Universal Robots PolyScope program: 33-trigger_reduced_mode.urp

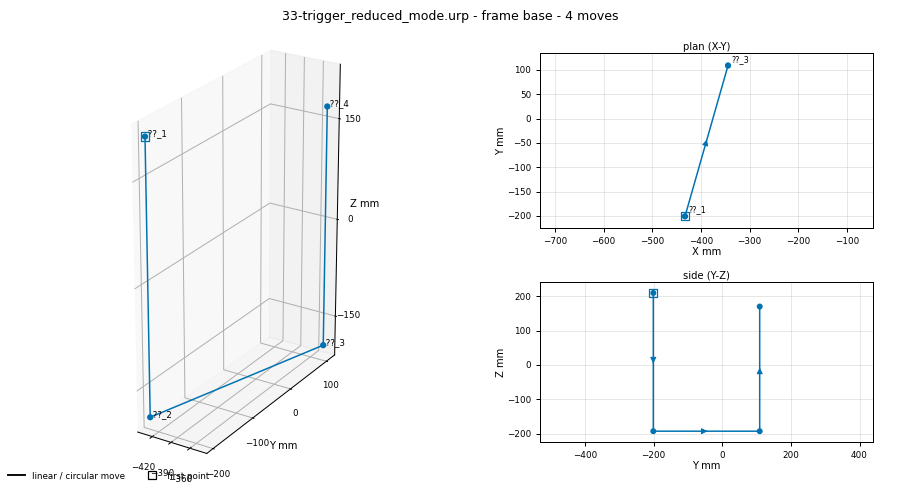
[picture p0: tool path of 33-trigger_reduced_mode.urp in frame base, 4 of 4 moves have a stored position in this frame; points joined in program order, loops and branches not executed]
ProgramRoot directory=/programs/usbdisk; kinematics=(a=[0.00023, -0.38811, -0.39243, -0.00016, 0.00019, 0], d=[0.08925, 195.22769, -194.66383, -0.45311, 0.09509, 0.08264], alpha=[1.57049, -0.00089, 0.00686, 1.56999, -1.56996, 0], deltaTheta=[-0.00001, -0.41907, 0.4289, -6.29306, -0.00007, 0], status=notLinearised); lastSavedInVersion=(project__name=Polyscope, major__version=3, minor__version=1, svn__revision=17141, build__date=Mar 06 2015, 07:52:30); name=33-trigger_reduced_mode; programVersion=(project__name=Polyscope, major__version=3, minor__version=1, svn__revision=17141, build__date=Mar 06 2015, 07:52:30); robotEnvironmentFileName=safty; serialNumberRobot=2014350456
  MainProgram cartesianAcceleration=1.2; cartesianSpeed=0.25; jointAcceleration=1.3962634015954636; jointSpeed=1.0471975511965976; sharedProcessMoveBlendRadius=0.025; motionType=JOINT_SPACE
    Move cartesianAcceleration=1.2; cartesianSpeed=0.25; jointAcceleration=1.3962634015954636; jointSpeed=1.0471975511965976; sharedProcessMoveBlendRadius=0.025; motionType=CARTESIAN_SPACE
      Waypoint blendRadius=0.05; cartesianAcceleration=1.2; cartesianSpeed=0.25; jointAcceleration=1.3962634015954636; jointSpeed=1.0471975511965976; nextMotionTime=2.0; stoppoint=true; useSharedBlendParameter=true; useSharedParameters=true; outputFlangePose=(pos=(x=-0.432847912452541, y=-0.20086659194210368, z=0.2098495284796807), rot=(x=-3.1225656389984957, y=0.16278110230970627, z=-0.16198721880946063)); position=TCP in base x=-432.85 y=-200.853 z=209.821 mm, rx=-3.1225 ry=0.1628 rz=-0.1621 rad; joints [-142.342, -96.295, -116.362, -62.279, 93.748, 133.656] deg; positionType=FIXED_POSITION; waypointPoseInFeatureCoordinates=(pos=(x=-0.4328500968425132, y=-0.20085347457033764, z=0.2098212918601961), rot=(x=-3.1224672981626562, y=0.1627652346722001, z=-0.162087261467964)); name=路点_1
      Waypoint blendRadius=0.05; cartesianAcceleration=1.2; cartesianSpeed=0.25; jointAcceleration=1.3962634015954636; jointSpeed=1.0471975511965976; nextMotionTime=2.0; stoppoint=true; useSharedBlendParameter=true; useSharedParameters=true; outputFlangePose=(pos=(x=-0.43284784754101663, y=-0.20086654166314177, z=-0.19296929807421476), rot=(x=-3.1225656377030893, y=0.1627811003512241, z=-0.16198721679836964)); position=TCP in base x=-432.87 y=-200.86 z=-192.961 mm, rx=-3.1226 ry=0.1627 rz=-0.1619 rad; joints [-142.362, -151.792, -117.864, -5.272, 93.408, 133.81] deg; positionType=FIXED_POSITION; waypointPoseInFeatureCoordinates=(pos=(x=-0.4328695456767533, y=-0.20086045026229912, z=-0.19296083589084112), rot=(x=-3.122584117311889, y=0.16271068994540802, z=-0.16187034783988982)); name=路点_2
      Waypoint blendRadius=0.05; cartesianAcceleration=1.2; cartesianSpeed=0.25; jointAcceleration=1.3962634015954636; jointSpeed=1.0471975511965976; nextMotionTime=2.0; stoppoint=true; useSharedBlendParameter=true; useSharedParameters=true; outputFlangePose=(pos=(x=-0.34441027168573285, y=0.10918607737217474, z=-0.19296936111808682), rot=(x=-3.1225656063558365, y=0.1627810982879899, z=-0.16198730339741577)); position=TCP in base x=-344.378 y=109.196 z=-192.994 mm, rx=-3.1226 ry=0.1628 rz=-0.1622 rad; joints [-179.766, -154.677, -134.205, 12.879, 89.614, 96.558] deg; positionType=FIXED_POSITION; waypointPoseInFeatureCoordinates=(pos=(x=-0.34437772167666364, y=0.10919607092421764, z=-0.1929939751957054), rot=(x=-3.122590823125009, y=0.1627656593988479, z=-0.16216513554717069)); name=路点_3
      Waypoint blendRadius=0.05; cartesianAcceleration=1.2; cartesianSpeed=0.25; jointAcceleration=1.3962634015954636; jointSpeed=1.0471975511965976; nextMotionTime=2.0; stoppoint=true; useSharedBlendParameter=true; useSharedParameters=true; outputFlangePose=(pos=(x=-0.3444101427544767, y=0.10918607791850427, z=0.17024960411493406), rot=(x=-3.122565609705968, y=0.16278110662614406, z=-0.16198730394031693)); position=TCP in base x=-344.41 y=109.18 z=170.245 mm, rx=-3.1226 ry=0.1627 rz=-0.162 rad; joints [-179.75, -83.836, -135.677, -56.488, 90.07, 96.448] deg; positionType=FIXED_POSITION; waypointPoseInFeatureCoordinates=(pos=(x=-0.3444101299808141, y=0.10917971943427503, z=0.17024457476537574), rot=(x=-3.122575244951181, y=0.16271155992446873, z=-0.16197719226190127)); name=路点_4
